(* IEC 61131-3 sources: RL_MAR/experiments/comparison/autoplc/results/qwen3.5-9b_20260511_180311/med_78, 1 file *)

(* ---- med_78_1.st ---- *)
FUNCTION_BLOCK RetractableRoofControl
VAR_INPUT
    RainSensor : BOOL;
    WindSensor : BOOL;
    TemperatureSensor : REAL;
END_VAR
VAR_OUTPUT
    RoofMotor : BOOL;
END_VAR
VAR
    Condition1 : BOOL;
    Condition2 : BOOL;
    Condition3 : BOOL;
END_VAR

Condition1 := RainSensor AND WindSensor;

IF Condition1 THEN
    RoofMotor := TRUE;
ELSIF RainSensor THEN
    RoofMotor := TRUE;
ELSIF TemperatureSensor < 20.0 THEN
    RoofMotor := TRUE;
ELSE
    RoofMotor := FALSE;
END_IF;

END_FUNCTION_BLOCK
